TYPE ST_System_MVHW_Parameter :
STRUCT
	AutoQuittierung			: BOOL;


END_STRUCT
END_TYPE

(* stored: Version 1.1.0.1, ProductVersion 3.1.4024.9
   DUT ST_System_MVHW_Parameter: Id {c081fe2e-593f-47be-876d-d055896c0e92} *)
